TYPE ST_Klima_Bueros :
STRUCT
	Temperatur			: REAL;
	Luftfeuchte_rel		: REAL;
END_STRUCT
END_TYPE

(* stored: Version 1.1.0.1, ProductVersion 3.1.4024.9
   DUT ST_Klima_Bueros: Id {653ca4c6-a82f-4e16-90e1-b42adc04d50c} *)
